% RSLogix 500 project ESTACION2.RSS, saved by version 8.40.00.08 %
PROJECT "UNTITLED"    % processor: MicroLogix 1500 %

PROGRAM FILES
  LAD 2   9 rungs

DATA FILES
  O0 OUTPUT  4 elements
  I1 INPUT  4 elements
  S2 STATUS  66 elements
  B3 BINARY  1 elements
  T4 TIMER  3 elements
  C5 COUNTER  1 elements
  R6 CONTROL  1 elements
  N7 INTEGER  1 elements
  F8 FLOAT  1 elements

LADDER 2
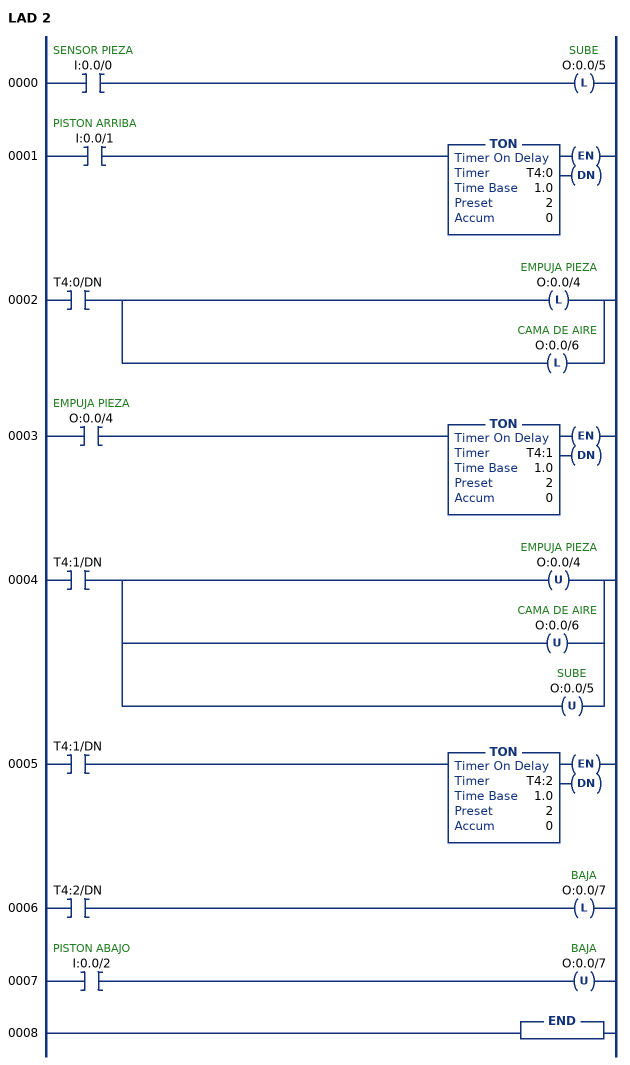
% Rung: 0 %
SOR XIC I:0.0/0 OTL O:0.0/5 EOR
%   I:0.0/0  "SENSOR PIEZA" %
%   O:0.0/5  "SUBE" %
% Rung: 1 %
SOR XIC I:0.0/1 TON T4:0 1.0 2 0 EOR
%   I:0.0/1  "PISTON ARRIBA" %
% Rung: 2 %
SOR XIC T4:0/DN BST OTL O:0.0/4 NXB OTL O:0.0/6 BND EOR
%   O:0.0/4  "EMPUJA PIEZA" %
%   O:0.0/6  "CAMA DE AIRE" %
% Rung: 3 %
SOR XIC O:0.0/4 TON T4:1 1.0 2 0 EOR
%   O:0.0/4  "EMPUJA PIEZA" %
% Rung: 4 %
SOR XIC T4:1/DN BST OTU O:0.0/4 NXB BST OTU O:0.0/6 NXB OTU O:0.0/5 BND BND EOR
%   O:0.0/4  "EMPUJA PIEZA" %
%   O:0.0/6  "CAMA DE AIRE" %
%   O:0.0/5  "SUBE" %
% Rung: 5 %
SOR XIC T4:1/DN TON T4:2 1.0 2 0 EOR
% Rung: 6 %
SOR XIC T4:2/DN OTL O:0.0/7 EOR
%   O:0.0/7  "BAJA" %
% Rung: 7 %
SOR XIC I:0.0/2 OTU O:0.0/7 EOR
%   I:0.0/2  "PISTON ABAJO" %
%   O:0.0/7  "BAJA" %
% Rung: 8 %
SOR END EOR

DATA TABLE (non-zero values as saved)
DATA T4
% .PRE .ACC %
% T4:0 % 2 0
% T4:1 % 2 0
% T4:2 % 2 0
